// TIA Portal V20 export
// export: Created 2026-04-11T06:02:29.7631224Z, ExportSetting WithDefaults, DisplayName Totally Integrated Automation Portal, DisplayVersion V20, DisplayName TIA Portal Openness, DisplayVersion V20, DisplayName TIA Portal Version Control Interface, DisplayVersion V20, DisplayName STEP 7 Professional, DisplayVersion V20, DisplayName STEP 7 Safety, DisplayVersion V20, DisplayName WinCC Basic/Comfort/Advanced, DisplayVersion V20, DisplayName WinCC Unified, DisplayVersion V20
TYPE "udtContC_C"
// stored: IsFailsafeCompliant false
   STRUCT
      COM_RST : Bool;
      MAN_ON : Bool;
      PVPER_ON : Bool;
      P_SEL : Bool;
      I_SEL : Bool;
      INT_HOLD : Bool;
      I_ITL_ON : Bool;
      D_SEL : Bool;
      CYCLE : Time;
      SP_INT : Real;
      PV_IN : Real;
      PV_PER : Word;
      MAN : Real;
      GAIN : Real;
      TI : Time;
      TD : Time;
      TM_LAG : Time;
      DEADB_W : Real;
      LMN_HLM : Real;
      LMN_LLM : Real;
      PV_FAC : Real;
      PV_OFF : Real;
      LMN_FAC : Real;
      LMN_OFF : Real;
      I_ITLVAL : Real;
      DISV : Real;
   END_STRUCT;
END_TYPE
